TYPE ST_ReceivedData :
STRUCT
	userId:	DINT;
	id:		DINT;
	title:	STRING(255);
	body:	STRING(255);
END_STRUCT
END_TYPE

(* stored: Version 1.1.0.1, ProductVersion 3.1.4024.3
   DUT ST_ReceivedData: Id {142a6d09-4e63-40d3-a899-c4fbb5d9d0c7} *)
